(* CODESYS project Interface Example.export

Project tree, tasks and I/O mapping:
  interface IMotor: Start, Stop, IsRunning
  program Main [ST]
  function block Motor [ST]: Start, Stop, IsRunning
*)

// IMotor
INTERFACE IMotor

METHOD Start : BOOL
VAR_INPUT
END_VAR
END_METHOD

METHOD Stop : BOOL
VAR_INPUT
END_VAR
END_METHOD

PROPERTY IsRunning : BOOL
GET
END_GET
SET
END_SET
END_PROPERTY

END_INTERFACE

// Main
PROGRAM Main
VAR_INPUT
	Motor : IMotor;
END_VAR


// Call a method
Motor.Start();

// Get a property
IF Motor.IsRunning THEN (**) END_IF

END_PROGRAM

// Motor
FUNCTION_BLOCK Motor IMPLEMENTS IMotor


// Motor control logic here

METHOD Start : BOOL
END_METHOD

METHOD Stop : BOOL
END_METHOD

PROPERTY IsRunning : BOOL
GET
END_GET
SET
END_SET
END_PROPERTY

END_FUNCTION_BLOCK
